{attribute 'linkalways'} 
{attribute 'no_explicit_call' := 'This FB is a CLASS and must be accessed using methods or properties'}
{attribute 'enable_dynamic_creation'}
FUNCTION_BLOCK Node_F_VN_SetAt_TcVnVector4_USINT EXTENDS VisionNode
VAR
    aElement : _TcVnVector4_USINT;
    ipContainer : _ITcVnContainer;
    nIndex : _ULINT(0);
    hrPrev : _HRESULT(S_OK);
    hresult : _HRESULT(S_OK);
END_VAR

METHOD PUBLIC  Clone : I_Node
VAR
	pNode : POINTER TO Node_F_VN_SetAt_TcVnVector4_USINT;
END_VAR
pNode := __NEW(Node_F_VN_SetAt_TcVnVector4_USINT);
Clone := pNode^;
END_METHOD

METHOD FB_init : BOOL
VAR_INPUT
	bInitRetains : BOOL; // if TRUE, the retain variables are initialized (warm start / cold start)
	bInCopyCode : BOOL;  // if TRUE, the instance afterwards gets moved into the copy code (online change)
END_VAR
AddInput('aElement', aElement);
AddInput('ipContainer', ipContainer);
AddParameter('nIndex', nIndex);
AddInput('hrPrev', hrPrev);
AddOutput('ipContainer', ipContainer);
AddOutput('hresult',hresult);
END_METHOD

METHOD PROTECTED OnExecute
hresult.Value := F_VN_SetAt_TcVnVector4_USINT(
    aElement := aElement.Value,
    ipContainer := ipContainer.Value,
    nIndex := nIndex.Value,
    hrPrev:= hrPrev.Value);
END_METHOD

METHOD PUBLIC PreExecutionCheck
VAR_INPUT
	Check : I_PreExecutionChecks;
END_VAR
Check.IsTrue(ipContainer.IsValid, 'ipContainer must be a valid container');
Check.IsTrue(ipContainer.IsType(TC_GLOBAL_CONST_LIST.ContainerType_Vector_TcVnVector4_USINT), 'ipContainer contains incorrect type');
END_METHOD

END_FUNCTION_BLOCK

(* stored: Version 1.1.0.1, ProductVersion 3.1.4026.13
   POU Node_F_VN_SetAt_TcVnVector4_USINT: Id {061c16ec-82eb-46dd-8b85-64c9484c094e}, SpecialFunc None
   Folder Constructor: Id {b3483091-f955-4ab4-bc83-a2f2c68a866b}
   Method Clone: Id {e88abb9c-aa22-4f2b-8061-7276534c19c9}
   Method FB_init: Id {138a7e2c-7bec-450d-84a1-6ac51c75a650}
   Method OnExecute: Id {da49ec29-b5b0-4edc-800c-e11af398de05}
   Method PreExecutionCheck: Id {1c031258-e63b-4ef5-9a87-d8a9af8c7a2e} *)
